PROGRAM main
VAR
	MainGreen : bool := True;
	MainYellow : bool := False;
	MainRed : bool := False;
	SideGreen : bool := False;
	SideYellow : bool := False;
	SideRed : bool := True;
	CarWaiting : bool := False;
	PedWaiting : bool := False;
	GreenTimer : TON;
	YellowTimer : TON;
	SideGreenTimer : TON;
	SideYellowTimer : TON;
END_VAR

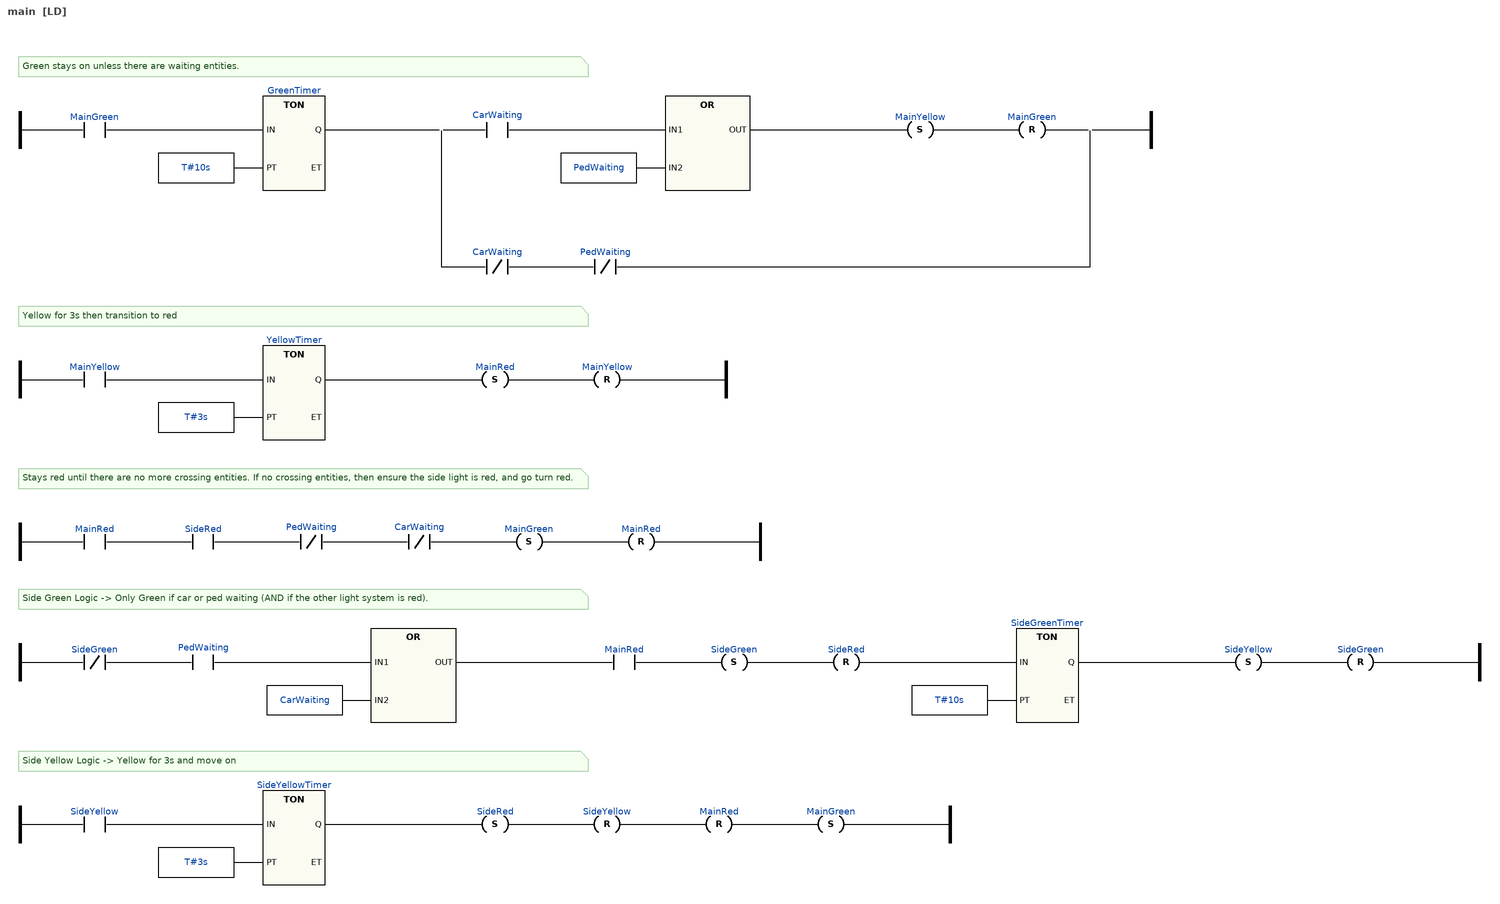
(* LD diagram, written out as Structured Text *)
(* Green stays on unless there are waiting entities. *)
GreenTimer(IN := MainGreen, PT := T#10s);
IF GreenTimer.Q AND CarWaiting OR PedWaiting THEN MainYellow := TRUE; END_IF;
IF GreenTimer.Q AND CarWaiting OR PedWaiting THEN MainGreen := FALSE; END_IF;
(* Yellow for 3s then transition to red *)
YellowTimer(IN := MainYellow, PT := T#3s);
IF YellowTimer.Q THEN MainRed := TRUE; END_IF;
IF YellowTimer.Q THEN MainYellow := FALSE; END_IF;
(* Stays red until there are no more crossing entities. If no crossing entities, then ensure the side light is red, and go turn red. *)
IF MainRed AND SideRed AND NOT PedWaiting AND NOT CarWaiting THEN MainGreen := TRUE; END_IF;
IF MainRed AND SideRed AND NOT PedWaiting AND NOT CarWaiting THEN MainRed := FALSE; END_IF;
(* Side Green Logic -> Only Green if car or ped waiting (AND if the other light system is red). *)
IF (NOT SideGreen AND PedWaiting OR CarWaiting) AND MainRed THEN SideGreen := TRUE; END_IF;
IF (NOT SideGreen AND PedWaiting OR CarWaiting) AND MainRed THEN SideRed := FALSE; END_IF;
SideGreenTimer(IN := (NOT SideGreen AND PedWaiting OR CarWaiting) AND MainRed, PT := T#10s);
IF SideGreenTimer.Q THEN SideYellow := TRUE; END_IF;
IF SideGreenTimer.Q THEN SideGreen := FALSE; END_IF;
(* Side Yellow Logic -> Yellow for 3s and move on *)
SideYellowTimer(IN := SideYellow, PT := T#3s);
IF SideYellowTimer.Q THEN SideRed := TRUE; END_IF;
IF SideYellowTimer.Q THEN SideYellow := FALSE; END_IF;
IF SideYellowTimer.Q THEN MainRed := FALSE; END_IF;
IF SideYellowTimer.Q THEN MainGreen := TRUE; END_IF;
(* drawn but not wired to any output: CarWaiting, PedWaiting *)
END_PROGRAM
